(* CODESYS project AstroBROT.library
   Title: AstroBROT
   Version: 0.3.0
   Placeholder: AstroBROT
   Company: BROT

Project tree, tasks and I/O mapping:
  libraries: Tc2_Math, * (Beckhoff Automation GmbH); Tc2_Standard, * (Beckhoff Automation GmbH); Tc2_System, * (Beckhoff Automation GmbH); Tc2_Utilities, * (Beckhoff Automation GmbH); Tc3_Module, * (Beckhoff Automation GmbH)
  DUTs/
    data type E_TestState
  GVLs/
  POUs/
    FUNCTION_BLOCKS/
      function block FB_ALTAZ2HADEC [ST]
      function block FB_CO_ABERRATION [ST]
      function block FB_CO_NUTATE [ST]
      function block FB_CO_REFRACT [ST]
      function block FB_EQ2HOR [ST]
      function block FB_HADEC2ALTAZ [ST]
      function block FB_HOR2EQ [ST]
      function block FB_NUTATE [ST]
      function block FB_PRECESS [ST]
      function block FB_SUNPOS [ST]
    FUNCTIONS/
      function ATAN2 [ST]
      function CO_REFRACT_FORWARD [ST]
      function CT2LST [ST]
      function DateTime2JD [ST]
      function JD2LST [ST]
      function POLY [ST]
      function TEN [ST]
    program MAIN [ST]
  VISUs/
*)

// DUTs/E_TestState
{attribute 'qualified_only'}
{attribute 'strict'}
TYPE E_TestState :
(
	IDLE,
	EQ2HOR,
	HOR2EQ,
	EQ2EQ,
	JD2LST,
	ERROR
);
END_TYPE

// POUs/FUNCTION_BLOCKS/FB_ALTAZ2HADEC
FUNCTION_BLOCK FB_ALTAZ2HADEC
VAR_INPUT
	alt			: LREAL;	// the local apparent altitude, in DEGREES
	az			: LREAL;	// the local apparent azimuth, in DEGREES
	lat			: LREAL;	// the local geodetic latitude, in DEGREES
END_VAR
VAR_OUTPUT
	ha			: LREAL;	// the local apparent hour angle, in DEGREES
	dec			: LREAL;	// the local apparent declination, in DEGREES
END_VAR
VAR
	alt_r		: LREAL;
	az_r		: LREAL;
	lat_r		: LREAL;
	sindec		: LREAL;
END_VAR
VAR CONSTANT
	d2r			: LREAL := PI/180.0;
	r2d			: LREAL := 180.0/PI;
	//h2r:	LREAL := PI/12.0;
	//h2d:	LREAL := 15.0;
END_VAR

(*https://github.com/wlandsman/IDLAstro/blob/master/pro/

  NAME:
    ALTAZ2HADEC
 PURPOSE:
    Convert Horizon (Alt-Az) coordinates to Hour Angle and Declination.
 EXPLANATION::
    Can deal with the NCP singularity.    Intended mainly to be used by
    program hor2eq.pro
 CALLING SEQUENCE:
   ALTAZ2HADEC, alt, az, lat, ha, dec

 INPUTS
   alt - the local apparent altitude, in DEGREES, scalar or vector
   az  - the local apparent azimuth, in DEGREES, scalar or vector,
         measured EAST of NORTH!!!  If you have measured azimuth west-of-south
        (like the book MEEUS does), convert it to east of north via:
                       az = (az + 180) mod 360

   lat -  the local geodetic latitude, in DEGREES, scalar or vector.

 OUTPUTS
   ha  -  the local apparent hour angle, in DEGREES.  The hour angle is the 
          time that right ascension of 0 hours crosses the local meridian.  
          It is unambiguously defined.
   dec -  the local apparent declination, in DEGREES.

 EXAMPLE:
     Arcturus is observed at an apparent altitude of 59d,05m,10s and an 
     azimuth (measured east of north) of 133d,18m,29s while at the 
     latitude of +43.07833 degrees.
     What are the local hour angle and declination of this object?

     IDL> altaz2hadec, ten(59,05,10), ten(133,18,29), 43.07833, ha, dec
     ===> Hour angle ha = 336.683 degrees
          Declination, dec = 19.1824 degrees

       The widely available XEPHEM code gets:
                 Hour Angle = 336.683
                 Declination = 19.1824

 REVISION HISTORY:
    Written  Chris O'Dell Univ. of Wisconsin-Madison May 2002*)

alt_r  := alt*d2r;
az_r := az*d2r;
lat_r := lat*d2r;

//******************************************************************************
// find local HOUR ANGLE (in degrees, from 0. to 360.)
ha := atan2( (-SIN(az_r)*COS(alt_r)), (-COS(az_r)*SIN(lat_r)*COS(alt_r)+SIN(alt_r)*COS(lat_r)));
ha := ha / d2r;
IF ha < 0.0 THEN 
	ha := ha + 360.0;
END_IF
 ha := MODABS(ha, 360.0);

// Find declination (positive if north of Celestial Equator, negative if south)
sindec := SIN(lat_r)*SIN(alt_r) + COS(lat_r)*COS(alt_r)*COS(az_r);
// convert dec to degrees
dec := ASIN(sindec)/d2r;

END_FUNCTION_BLOCK

// POUs/FUNCTIONS/TEN
FUNCTION TEN : LREAL
VAR_INPUT
	dd, mm, ss	: LREAL;
END_VAR
VAR
END_VAR

TEN := dd + (mm/60.0) + (ss/3600.0);

END_FUNCTION

// POUs/FUNCTIONS/ATAN2
FUNCTION ATAN2 : LREAL
VAR_INPUT
	y		: LREAL;
	x		: LREAL;
END_VAR
VAR
END_VAR

(* source: https://de.wikipedia.org/wiki/Arctan2 *)
ATAN2 := 0.0;

IF x > 0 THEN
	ATAN2 := ATAN(y/x);
ELSIF x < 0 AND y > 0 THEN
	ATAN2 := ATAN(y/x) + PI;
ELSIF x < 0 AND y = 0 THEN
	ATAN2 := PI;
ELSIF x < 0 AND y < 0 THEN
	ATAN2 := ATAN(y/x) - PI;
ELSIF x = 0 AND y > 0 THEN
	ATAN2 := PI/2.0;
ELSIF x = 0 AND y < 0 THEN
	ATAN2 := -PI/2.0;
END_IF

END_FUNCTION

// POUs/FUNCTION_BLOCKS/FB_CO_ABERRATION
FUNCTION_BLOCK FB_CO_ABERRATION
VAR_INPUT
	jd			: LREAL;		// Julian Date
	ra			: LREAL;		// RA in degrees
	dec			: LREAL; 		// Dec in degrees
	eps 		: LREAL := 0.0;
END_VAR
VAR_OUTPUT
	d_ra		: LREAL;
	d_dec		: LREAL;
END_VAR
VAR
	sunpos		: FB_SUNPOS;
	nutate		: FB_NUTATE;
	sunra		: LREAL;
	sundec		: LREAL;
	sunlon		: LREAL;
	d_psi		: LREAL;
	d_epsilon	: LREAL; 
	eps0		: LREAL;
	t, e, peri, cd, sd, ce, te, cp, sp, cs, ss, ca, sa, term1, term2, term3, term4: LREAL;
END_VAR
VAR CONSTANT
	d2r 		: LREAL := PI/180.0;
	k			: LREAL := 20.49552; 	//constant of aberration, in arcseconds
	
END_VAR

(* https://github.com/wlandsman/IDLAstro/blob/master/pro/co_aberration.pro
;+
;  NAME:
;     CO_ABERRATION
; PURPOSE:
;     Calculate changes to Ra and Dec due to the effect of annual aberration 
; EXPLANATION:
;      as described in Meeus, Chap 23.
; CALLING SEQUENCE:
;      co_aberration, jd, ra, dec, d_ra, d_dec, [EPS = ]
; INPUTS
;       jd      : Julian Date [scalar or vector]
;       ra, dec : ra  and dec's in degrees
;
; OUTPUTS
;       d_ra, d_dec: the corrections to ra and dec due to aberration in 
;                    degrees.  (These values can be added to the true RA 
;                    and dec to get the apparent position).   Note that d_ra
;                     is *not* multiplied by cos(dec), so that 
;                     apparent_ra = ra + d_ra. 
; OPTIONAL INPUT KEYWORD:
;       eps : set this to the true obliquity of the ecliptic (in radians), or
;         it will be set for you if you don't know it (in that case, set it to
;                 an empty variable).
; NOTES:
;  These formula are from Meeus, Chapters 23.  Accuracy is much better than 1 
;   arcsecond.
;
;   The maximum deviation due to annual aberration is 20.49" and occurs when the
;   Earth velocity is perpendicular to the direction of the star.
;
; REVISION HISTORY:
;   Written, June 2002,      Chris O'Dell, U. of Wisconsin
;   Fix error with vector input   W. Landsman   June 2009
;   June 2009 update fixed case where JD was scalar but RA,Dec were vectors, but 
;     broke the case when both JD and RA,Dec were vectors Aug 2012 W. Landsman
;   Further fix when JD is 1 element vector  W. Landsman
;
;	UPDATE: HAS BEEN REWORKED FOR THE COORD STRUCTURE -> OUTPUT IS IN DEGREES
*)

T := (jd -2451545.0)/36525.0; // julian centuries from J2000 of jd.

IF eps = 0.0 THEN
	// must calculate obliquity of ecliptic
	nutate(jd := jd, nut_long => d_psi, nut_obliq => d_epsilon); //d_psi and d_epsilon in degrees
	eps0 := ten(23,26,21.448)*3600.0 - 46.8150*T - 0.00059*EXPT(T, 2) +  0.001813*EXPT(T, 3);
	// TRUE obliquity OF the ecliptic in radians
	eps := (eps0 + d_epsilon)/3600.0*d2r; 	
END_IF

sunpos(jd := jd, ra => sunra, dec => sundec, longmed => sunlon);

// Earth's orbital eccentricity
e := 0.016708634 - 0.000042037*T - 0.0000001267*EXPT(T, 2);
// longitude of perihelion, in degrees 
peri := 102.93735 + 1.71946*T + 0.00046*EXPT(T, 2);

//Useful Trig Functions
cd := COS(dec*d2r);		sd := SIN(dec*d2r);
ce := COS(eps); 		te := TAN(eps);
cp := COS(peri*d2r);	sp := SIN(peri*d2r);
cs := COS(sunlon*d2r);	ss := SIN(sunlon*d2r);
ca := COS(ra*d2r);		sa := SIN(ra*d2r);

term1 := (ca*cs*ce + sa*ss)/cd;
term2 := (ca*cp*ce + sa*sp)/cd;
term3 := (cs*ce*(te*cd - sa*sd) + ca*sd*ss);
term4 := (cp*ce*(te*cd - sa*sd) + ca*sd*sp);

d_ra := (-k * term1 + e*k * term2)/3600;
d_dec := (-k * term3 + e*k * term4)/3600;

END_FUNCTION_BLOCK

// POUs/FUNCTION_BLOCKS/FB_SUNPOS
FUNCTION_BLOCK FB_SUNPOS
VAR_INPUT
	jd				: LREAL;		// Julian Date
END_VAR
VAR_OUTPUT
	ra				: LREAL;		// right ascension
	dec				: LREAL;		// declination of the sun 
	longmed			: LREAL;		// longitude
	oblt			: LREAL;		// True Obliquity
END_VAR
VAR
	t				: LREAL;		//  Julian centuries FROM 1900.0
	l				: LREAL;		//  sun's mean longitude
	me				: LREAL;		// Earth's mean anomaly
	ellcor			: LREAL;		// ellipticity of the orbit
	mv				: LREAL;		// mean anomaly of Venus
	vencorr			: LREAL;		
	mm				: LREAL;		
	marscorr		: LREAL;		
	mj				: LREAL;		
	jupcorr			: LREAL;		
	d				: LREAL;		
	longterm		: LREAL;		
	mooncorr		: LREAL;		
	omega			: LREAL;
END_VAR
VAR CONSTANT
	d2r				: LREAL := PI/180.0; // Pi/180
END_VAR

(* https://github.com/wlandsman/IDLAstro/blob/master/pro/
NOTES:
;       Patrick Wallace (Rutherford Appleton Laboratory, UK) has tested the
;       accuracy of a C adaptation of the sunpos.pro code and found the 
;       following results.   From 1900-2100 SUNPOS  gave 7.3 arcsec maximum 
;       error, 2.6 arcsec RMS.  Over the shorter interval 1950-2050 the figures
;       were 6.4 arcsec max, 2.2 arcsec RMS.  
;
;       The returned ra and Dec are in the given date's equinox.
;
;       Procedure was extensively revised in May 1996, and the new calling
;       sequence is incompatible with the old one.source: https://idlastro.gsfc.nasa.gov/ftp/pro/astro/sunpos.pro *)

//  form TIME in Julian centuries FROM 1900.0
t := (jd - 2415020.0) / 36525.0;

//  form sun's mean longitude
l := (279.696678 + LMOD(36000.768925 * t, 360.0)) * 3600.0;

//  allow for ellipticity of the orbit (equation of centre) using the Earth's mean anomaly ME
me := 358.475844 + LMOD(35999.049750 * t, 360.0);
ellcor  := (6910.1 - 17.2 * t) * SIN(me * d2r) + 72.3 * SIN(2.0 * me*d2r);
l := l + ellcor;
 
// allow FOR the Venus perturbations using the mean anomaly OF Venus MV
mv := 212.603219 + LMOD(58517.803875 * t, 360.0);
vencorr := 4.8 * COS((299.1017 + mv - me)*d2r) + 
           5.5 * COS((148.3133 +  2.0 * mv  -  2.0 * me )*d2r) + 
           2.5 * COS((315.9433 +  2.0 * mv  -  3.0 * me )*d2r) + 
           1.6 * COS((345.2533 +  3.0 * mv  -  4.0 * me )*d2r) + 
           1.0 * COS((318.15   +  3.0 * mv  -  5.0 * me )*d2r);
l := l + vencorr;

//  Allow FOR the Mars perturbations using the mean anomaly OF Mars MM
mm := 319.529425  +  LMOD( 19139.858500 * t,  360.0 );
marscorr := 2.0 * COS((343.8883 -  2.0 * mm  +  2.0 * me)*d2r ) + 
            1.8 * COS((200.4017 -  2.0 * mm  + me) * d2r);
l := l + marscorr;

// Allow FOR the Jupiter perturbations using the mean anomaly OF Jupiter MJ
mj := 225.328328  +  LMOD( 3034.6920239 * t,  360.0 );
jupcorr := 7.2 * COS(( 179.5317 - mj + me )*d2r) + 
           2.6 * COS((263.2167  -  MJ ) *d2r) + 
           2.7 * COS(( 87.1450  -  2.0 * mj  +  2.0 * me ) *d2r) + 
           1.6 * COS((109.4933  -  2.0 * mj  +  me ) *d2r);
l := l + jupcorr;

// Allow FOR the Moons perturbations using the mean elongation OF the Moon from the Sun D
d := 350.7376814  + LMOD(445267.11422 * t,  360.0);
mooncorr  := 6.5 * SIN(d * d2r);
l := l + mooncorr;

// Allow for long period terms
longterm := 6.4 * SIN((231.19  +  20.20 * t) * d2r);
l :=  l + longterm;
l :=  LMOD(l + 2592000.0,  1296000.0); 
longmed := l / 3600.0;

// Allow for Aberration
l :=  l - 20.5;

// Allow for Nutation using the longitude of the Moons mean node OMEGA
omega := 259.183275 - LMOD(1934.142008 * t, 360.0);
l :=  l - 17.2 * SIN(omega * d2r);

// Form the True Obliquity
oblt := 23.452294 - 0.0130125 * t + (9.2 * COS(omega * d2r)) / 3600.0;

// Form Right Ascension AND Declination
l := l / 3600.0;
ra := ATAN2(SIN(l * d2r) * COS(oblt * d2r), COS(l * d2r));
dec := ASIN(SIN(l * d2r) * SIN(oblt * d2r));
 
ra := ra/d2r;
ra := MODABS(ra, 360.0);
dec := dec/d2r;

END_FUNCTION_BLOCK

// POUs/FUNCTION_BLOCKS/FB_NUTATE
FUNCTION_BLOCK FB_NUTATE
VAR_INPUT
	jd				: LREAL;			// Julian date
END_VAR
VAR_OUTPUT
	nut_long		: LREAL := 0.0;
	nut_obliq		: LREAL := 0.0;
END_VAR
VAR
	t				: LREAL;
	d, M, Mprime, F, omega: LREAL;
	arg, sarg, carg	: ARRAY[0..62] OF LREAL;
	I				: INT;
END_VAR
VAR CONSTANT
	d2r				: LREAL := PI/180.0;
	coeff1			: ARRAY[0..3] OF LREAL := [297.85036, 445267.111480, -0.0019142,  1.0/189474];
	coeff2			: ARRAY[0..3] OF LREAL := [357.52772,  35999.050340, -0.0001603, -1.0/3E5]; 
	coeff3			: ARRAY[0..3] OF LREAL := [134.96298, 477198.867398,  0.0086972,  1.0/5.625E4]; 
	coeff4			: ARRAY[0..3] OF LREAL :=  [93.27191, 483202.017538, -0.0036825, -1.0/3.27270E5]; 
  	coeff5			: ARRAY[0..3] OF LREAL := [125.04452,  -1934.136261,  0.0020708,  1.0/4.5E5];
	d_lng			: ARRAY[0..62] OF LREAL := [0,-2,0,0,0,0,-2,0,0,-2,-2,-2,0,2,0,2,0,0,-2,0,2,0,0,-2,0,-2,0,0,2,-2,0,-2,0,0,2,2,0,-2,0,2,2,-2,-2,2,2,0,-2,-2,0,-2,-2,0,-1,-2,1,0,0,-1,0,0,2,0,2]; 
	m_lng			: ARRAY[0..62] OF LREAL := [0,0,0,0,1,0,1,0,0,-1,17(0),2,0,2,1,0,-1,0,0,0,1,1,-1,0,0,0,0,0,0,-1,-1,0,0,0,1,0,0,1,0,0,0,-1,1,-1,-1,0,-1];
	mp_lng			: ARRAY[0..62] OF LREAL := [0,0,0,0,0,1,0,0,1,0,1,0,-1,0,1,-1,-1,1,2,-2,0,2,2,1,0,0,-1,0,-1,0,0,1,0,2,-1,1,0,1,0,0,1,2,1,-2,0,1,0,0,2,2,0,1,1,0,0,1,-2,1,1,1,-1,3,0];
	f_lng			: ARRAY[0..62] OF LREAL := [0,2,2,0,0,0,2,2,2,2,0,2,2,0,0,2,0,2,0,2,2,2,0,2,2,2,2,0,0,2,0,0,0,-2,2,2,2,0,2,2,0,2,2,0,0,0,2,0,2,0,2,-2,0,0,0,2,2,0,0,2,2,2,2];
	om_lng			: ARRAY[0..62] OF LREAL := [1,2,2,2,0,0,2,1,2,2,0,1,2,0,1,2,1,1,0,1,2,2,0,2,0,0,1,0,1,2,1,1,1,0,1,2,2,0,2,1,0,2,1,1,1,0,1,1,1,1,1,0,0,0,0,0,2,0,0,2,2,2,2];
	sin_lng			: ARRAY[0..62] OF LREAL := [-171996, -13187, -2274, 2062, 1426, 712, -517, -386, -301, 217, -158, 129, 123, 63, 63, -59, -58, -51, 48, 46, -38, -31, 29, 29, 26, -22, 21, 17, 16, -16, -15, -13, -12, 11, -10, -8, 7, -7, -7, -7, 6,6,6,-6,-6,5,-5,-5,-5,4,4,4,-4,-4,-4,3,-3,-3,-3,-3,-3,-3,-3 ];
	sdelt			: ARRAY[0..62] OF LREAL := [-174.2, -1.6, -0.2, 0.2, -3.4, 0.1, 1.2, -0.4, 0, -0.5, 0, 0.1, 0,0,0.1, 0,-0.1,10(0), -0.1, 0, 0.1, 33(0)];
	cos_lng			: ARRAY[0..62] OF LREAL := [ 92025, 5736, 977, -895, 54, -7, 224, 200, 129, -95,0,-70,-53,0, -33, 26, 32, 27, 0, -24, 16,13,0,-12,0,0,-10,0,-8,7,9,7,6,0,5,3,-3,0,3,3, 0,-3,-3,3,3,0,3,3,3, 14(0)] ;
	cdelt			: ARRAY[0..62] OF LREAL := [8.9, -3.1, -0.5, 0.5, -0.1, 0.0, -0.6, 0.0, -0.1, 0.3, 53(0)];
END_VAR

//https://github.com/wlandsman/IDLAstro/blob/master/pro/nutate.pro
(*METHOD:
;       Uses the formula in Chapter 22 of ``Astronomical Algorithms'' by Jean 
;       Meeus (1998, 2nd ed.) which is based on the 1980 IAU Theory of Nutation
;       and includes all terms larger than 0.0003".*)

//  form time in Julian centuries from 1900.0

t := (jd - 2451545.0)/36525.0;

// Mean elongation of the Moon

d := poly(T, coeff1)*d2r;
d := MODABS(d, 2.0*PI);

// Sun's mean anomaly

M := poly(T,coeff2)*d2r;
M := MODABS(M, 2.0*PI);

// Moon's mean anomaly

Mprime := poly(T,coeff3)*d2r;
Mprime := MODABS(Mprime, 2.0*PI);

// Moon's argument of latitude

F := poly(T, coeff4 )*d2r;
F := MODABS(F, 2.0*PI);

// Longitude OF the ascending node OF the Moon's mean orbit on the ecliptic,
//  measured from the mean equinox of the date

omega := poly(T, coeff5)*d2r;
omega := MODABS(omega, 2.0*PI);


// Sum the periodic terms 
FOR i:=0 TO 62 DO
	arg[i] := d_lng[i]*d + m_lng[i]*m +mp_lng[i]*mprime + f_lng[i]*f +om_lng[i]*omega;
	sarg[i] := SIN(arg[i]);
	carg[i] := COS(arg[i]);
END_FOR

nut_long  := 0.0;
nut_obliq := 0.0;

FOR i:=0 TO 62 DO
	nut_long  := nut_long  + 0.0001*( (sdelt[i]*t + sin_lng[i])*sarg[i]);
	nut_obliq := nut_obliq + 0.0001*( (cdelt[i]*t + cos_lng[i])*carg[i]);
END_FOR

END_FUNCTION_BLOCK

// POUs/FUNCTIONS/POLY
FUNCTION POLY : LREAL
VAR_INPUT
	X			: LREAL;
	COEFFS		: ARRAY [0..3] OF LREAL;
END_VAR
VAR
END_VAR

POLY := COEFFS[0]*EXPT(X, 0) + COEFFS[1]*EXPT(X, 1) + COEFFS[2]*EXPT(X, 2) + COEFFS[3]*EXPT(X, 3);

END_FUNCTION

// POUs/FUNCTION_BLOCKS/FB_CO_NUTATE
FUNCTION_BLOCK FB_CO_NUTATE
VAR_INPUT
	jd			: LREAL;		// Julian date
	ra			: LREAL;		// RA in degrees
	dec			: LREAL;		// Dec in degrees
END_VAR
VAR_OUTPUT
	d_ra		: LREAL;		// RA diff in degrees
	d_dec		: LREAL;		// Dec diff in degrees
	eps			: LREAL;		// TRUE obliquity OF the ecliptic in radians
	d_psi		: LREAL;		// in arcsec
	d_eps		: LREAL;
END_VAR
VAR
	T, eps0, ce, se,x,y,z,x2,y2,z2,rad,xyproj,ra2,dec2: LREAL;
	nutate		: FB_NUTATE;
END_VAR
VAR CONSTANT
	d2r			: LREAL := PI/180.0;
	d2as		: LREAL := PI/(180.0*3600.0);
END_VAR

// https://github.com/wlandsman/IDLAstro/blob/master/pro/co_nutate.pro
(*EXPLANATION:
;     Calculates necessary changes to ra and dec due to
;     the nutation of the Earth's rotation axis, as described in Meeus, Chap 23.
;     Uses formulae from Astronomical Almanac, 1984, and does the calculations
;     in equatorial rectangular coordinates to avoid singularities at the
;     celestial poles.*)
// Julian centuries FROM J2000 OF jd.
T := (jd -2451545.0)/36525.0; 

// must calculate obliquity OF ecliptic
nutate(jd := jd,
		nut_long => d_psi, 
		nut_obliq => d_eps); 

eps0 := 23.4392911*3600.0 - 46.8150*T - 0.00059*EXPT(T, 2) + 0.001813*EXPT(T, 3);
eps := (eps0 + d_eps)/3600.0*d2r; // TRUE obliquity OF the ecliptic in radians
 
//useful numbers
ce := COS(eps);
se := SIN(eps);

// convert ra-dec to equatorial rectangular coordinates
x := COS(ra*d2r) * COS(dec*d2r);
y := SIN(ra*d2r) * COS(dec*d2r);
z := SIN(dec*d2r);

// apply corrections to each rectangular coordinate
x2 := x - (y*ce + z*se)*d_psi * d2as;
y2 := y + (x*ce*d_psi - z*d_eps) * d2as;
z2 := z + (x*se*d_psi + y*d_eps) * d2as;

// convert back to equatorial spherical coordinates
rad := SQRT(x2*x2 + y2*y2 + z2*z2);
xyproj := SQRT(x2*x2 + y2*y2);

ra2  := x2 * 0.0;
dec2 := x2 * 0.0;

// Calculate Ra and Dec in RADIANS (later convert to DEGREES)
IF (xyproj = 0) AND (z <> 0) THEN
	// places where xyproj=0 (point at NCP or SCP)
	dec2 := ASIN(z2/rad);
	ra2 := 0.0;
END_IF
 
IF (xyproj <> 0) THEN
	// places other than NCP or SCP
	ra2 := ATAN2(y2, x2);
	dec2 := ASIN(z2/rad);
END_IF

// convert to DEGREES

ra2 := ra2 /d2r;
dec2 := dec2 /d2r;

ra2 := MODABS(ra2, 360.0);


// Return changes in ra and dec
d_ra := (ra2 - ra);
d_dec := (dec2 - dec);

END_FUNCTION_BLOCK

// POUs/FUNCTION_BLOCKS/FB_CO_REFRACT
FUNCTION_BLOCK FB_CO_REFRACT
VAR_INPUT
	old_alt			: LREAL;			// old alt in degrees
	altitude		: LREAL := 0.0;		// altitude of observatory
	pressure		: LREAL := 0.0;		// pressure
	temperature		: LREAL := 0.0;		// temperature
	epsilon			: LREAL := 0.25; 	//accuracy of iteration for observed=TRUE case, in arcseconds
	TO_OBSERVED		: BOOL;
END_VAR
VAR_OUTPUT
	new_alt			: LREAL;
END_VAR
VAR
	aout, P, T, dr, cur, last : LREAL;
END_VAR
VAR CONSTANT
	alpha 			: LREAL := 0.0065; 	//temp lapse rate [deg C per meter]
END_VAR

// https://github.com/wlandsman/IDLAstro/blob/master/pro/co_refract.pro
IF temperature = 0.0 THEN
	IF altitude > 11000.0 THEN 
		temperature := 211.5; 
	ELSE 
		temperature := 283.0 - alpha*altitude;
	END_IF
END_IF

// estimate Pressure based on altitude, using U.S. Standard Atmosphere formula.
IF pressure = 0 THEN 
	pressure := 1010.0*EXPT(1-6.5/288000*altitude, 5.255);
END_IF

IF NOT TO_OBSERVED THEN 
	aout := old_alt - co_refract_forward(old_alt, P:=pressure,T:=temperature);
ELSE
	aout := 0.0;
	P := pressure; T := temperature;
	//calculate initial refraction guess
	dr := co_refract_forward(old_alt, P:=P, T:=T);
	cur := old_alt + dr; // guess of observed location

	REPEAT 
	 	last := cur;
		dr := co_refract_forward(cur, P:= P, T:=T);
	  	cur := old_alt + dr;
	UNTIL ABS(last-cur)*3600.0 < epsilon
	END_REPEAT
	aout := cur;
END_IF

new_alt := aout;

END_FUNCTION_BLOCK

// POUs/FUNCTIONS/CO_REFRACT_FORWARD
FUNCTION CO_REFRACT_FORWARD : LREAL
VAR_INPUT
	a			: LREAL; 			// The observed (apparent) altitude, in DEGREES.
	P			: LREAL := 1010.0;	// Pressure [in millibars]. Default is 1010 millibars.
	T			: LREAL := 0.0;		// Ground Temp [in Celsius].  Default is 0 Celsius.
END_VAR
VAR
	ref			: LREAL;
	tpcor		: LREAL;
END_VAR
VAR CONSTANT
	d2r 		: LREAL := PI/180.0;
END_VAR

a := LIMIT(0.0, a, 90.0);
P := LIMIT(600.0, P, 1200.0);
T := LIMIT(-40.0, T, 40.0);

IF a >= 15.0 THEN
	ref := 1.0 / TAN((a + 7.31 / (a + 4.4)) * d2r);
ELSE
	ref := 3.569 * (0.1594 + 0.0196 * a + 0.00002 * EXPT(a, 2)) / (1.0 + 0.505 * a + 0.0845 * EXPT(a, 2));
END_IF
tpcor := P * 283.15 / (1010.0 * (273.15 + T));
CO_REFRACT_FORWARD := tpcor * ref;

END_FUNCTION

// POUs/FUNCTION_BLOCKS/FB_EQ2HOR
FUNCTION_BLOCK FB_EQ2HOR
VAR_INPUT
	ra				: LREAL;	// right ascension in degrees
	dec				: LREAL;	// declination in degrees
	jd				: LREAL;	// Julian Date
	lon				: LREAL;	// longitude in degrees
	lat				: LREAL;	// latitude in degrees
	ws				: BOOL := FALSE; 	// Set this to TRUE get the azimuth measured westward FROM south (NOT East of North).
	precess			: BOOL := TRUE; 	// Set this to 1 to force precession [default], 0 for no precession correction
	nutate			: BOOL := TRUE; 	// Set this to 1 to force nutation [default], 0 for no nutation correction.
	aberration		: BOOL := TRUE; 	// Set this to 1 to force aberration correction [default], 0 for no correction.
	refract 		: BOOL := TRUE; 	// Set to 1 to force refraction correction[default] (for actual sky coord), 0 for no correction (for theoretical coord).
	refract_to_observed : BOOL := TRUE;
	altitude		: LREAL := 0.0;
END_VAR
VAR_OUTPUT
	alt				: LREAL;		// altitude in degrees
	az				: LREAL;		// azimuth in degrees
	ha				: LREAL;		// hour angle in degreesss
END_VAR
VAR
	tstart, J_now	: LREAL;
	lmst			: LREAL;
	last			: LREAL;
	d_psi			: LREAL;
	eps				: LREAL;
	fbprecess		: FB_PRECESS;
	hadec2altaz		: FB_HADEC2ALTAZ;
	co_nutate		: FB_CO_NUTATE;
	co_aberration	: FB_CO_ABERRATION;
	co_refract		: FB_CO_REFRACT;
	ra_pre			: LREAL;		// Precessed RA in degrees
	dec_pre			: LREAL;		// Precessed Dec in degrees
	d_ra_abr		: LREAL;		// Difference in RA due to aberration
	d_dec_abr		: LREAL;		// Difference in Dec due to aberration
	d_ra_nut		: LREAL;		// Difference in RA due to nutation
	d_dec_nut		: LREAL;		// Difference in Dec due to nutation
END_VAR
VAR CONSTANT
	// easier then functions
	d2r				: LREAL := PI/180.0;
	h2r				: LREAL := PI/12.0;
	jd2000			: LREAL := 2451545.0;
END_VAR

(* source https://github.com/wlandsman/IDLAstro/blob/master/pro/eq2hor.pro 

PURPOSE:
	Convert celestial  (ra-dec) coords to local horizon coords (alt-az).

DESCRIPTION:
This  code calculates horizon (alt,az) coordinates from equatorial
(ra,dec) coords. It is typically accurate to about 1 arcsecond or better (I
have checked the output against the publicly available XEPHEM software). It
performs precession, nutation, aberration, and refraction corrections. [...]
*)


tstart := 2000.0;

(* ******************************************************************************
 PRECESS coordinates to current date
 (uses astro lib procedure PRECESS.pro)
*)
J_now := (JD - jd2000)/365.25 + 2000.0; // compute current equinox
IF precess THEN
	fbprecess( 
		ra := ra, 
		dec := dec, 
		equinox1 := tstart, 
		equinox2 := J_now, 
		ra_precessed => ra_pre, 
		dec_precessed => dec_pre);
ELSE
	ra_pre := ra;
	dec_pre := dec;
END_IF

(******************************************************************************
 calculate NUTATION and ABERRATION Corrections to Ra-Dec 
*)

IF nutate THEN
	co_nutate(	
		jd := jd, 
		ra := ra_pre, 
		dec := dec_pre, 
		d_ra => d_ra_nut, 
		d_dec => d_dec_nut,
		eps=>eps, 
		d_psi=>d_psi);
END_IF

IF ABERRATION THEN	
	co_aberration(	
		jd := jd, 
		ra := ra_pre, 
		dec := dec_pre, 
		d_ra => d_ra_abr, 
		d_dec => d_dec_abr,
		eps := eps);	
END_IF
ra := ra_pre + d_ra_abr + d_ra_nut;
dec := dec_pre + d_dec_abr + d_dec_nut;

(***************************************************************************************
Calculate LOCAL MEAN SIDEREAL TIME *)
lmst := jd2lst(JD:=jd, lon:=lon);
// calculate local APPARENT sidereal time
last := lmst + d_psi *COS(eps)/3600.0 ; //add correction in degrees

(******************************************************************************
 Find hour angle (in DEGREES) *)
ha := last - ra;
ha := MODABS(ha, 360.0);

(*******************************************************************************
 Now do the spherical trig to get APPARENT alt,az. *)
hadec2altaz(	
	ha := ha, 
	dec := dec, 
	lat := lat, 
	alt => alt, 
	az => az, 
	WS := WS);

(********************************************************************************************
 Make Correction for ATMOSPHERIC REFRACTION
 (use this for visible and radio wavelengths; author is unsure about other wavelengths.
  See the comments in CO_REFRACT for more details.) *)
IF refract THEN 
	co_refract(	
		old_alt := alt, 
		altitude := altitude, 
		to_observed := refract_to_observed, 
		new_alt => alt);
END_IF

END_FUNCTION_BLOCK

// POUs/FUNCTIONS/JD2LST
FUNCTION JD2LST : LREAL
VAR_INPUT
	jd			: LREAL;	// Julian date
	lon			: LREAL;	// longitude in degrees
END_VAR
VAR
	T			: LREAL;
	theta0		: LREAL;
END_VAR
VAR CONSTANT
	jd2000		: LREAL := 2451545.0;
END_VAR

// following https://squarewidget.com/astronomical-calculations-sidereal-time/
T := ((jd - jd2000) / 36525.0);
theta0 := 280.46061837 + 360.98564736629 * (JD - jd2000) + (0.000387933 * T * T) - (T * T * T / 38710000.0); // (12.4)

// LST is only defined from 0 to 360
JD2LST := MODABS(theta0 + lon, 360.0); // LST in degrees

END_FUNCTION

// POUs/FUNCTION_BLOCKS/FB_PRECESS
FUNCTION_BLOCK FB_PRECESS
VAR_INPUT
	ra				: LREAL;		// RA in degrees
	dec				: LREAL;		// Dec in degrees
	equinox1		: LREAL;
	equinox2		: LREAL;
END_VAR
VAR_OUTPUT
	ra_precessed	: LREAL;
	dec_precessed	: LREAL;
END_VAR
VAR
	ra_rad			: LREAL;		// RA in rad
	dec_rad			: LREAL;		// Dec in rad
	a, b, c, t		: LREAL;
	x, x2			: ARRAY[0..2] OF LREAL;
	st1				: LREAL;
	rot				: ARRAY[0..2,0..2] OF LREAL;
	sina, sinb, sinc, cosa,cosb,cosc: LREAL;
END_VAR
VAR CONSTANT
	d2r 			: LREAL := PI/180.0;
	sec_to_rad 		: LREAL := d2r/3600.0;
END_VAR

//https://github.com/wlandsman/IDLAstro/blob/master/pro/precess.pro

(*
; RESTRICTIONS:
;       Accuracy of precession decreases for declination values near 90 
;       degrees.  PRECESS should not be used more than 2.5 centuries from
;       2000 on the FK5 system (1950.0 on the FK4 system).
; PROCEDURE:
;       Algorithm from Computational Spherical Astronomy by Taff (1983), 
;       p. 24. (FK4). FK5 constants from "Astronomical Almanac Explanatory
;       Supplement 1992, page 104 Table 3.211.1.
*)

// deg 2 radian
ra_rad := ra*d2r;
dec_rad := dec*d2r;


a := COS( dec_rad );
x[0] := a*COS(ra_rad); x[1] := a*SIN(ra_rad); x[2] := SIN(dec_rad);

//*** PREMAT code starts here
ST1 := 0.001*( equinox1 - 2000.0);
t := 0.001*( equinox2 - equinox1);
//  Compute 3 rotation angles
A := sec_to_rad * T * (23062.181 + ST1*(139.656 +0.0139*ST1) + T*(30.188 - 0.344*ST1+17.998*T));
B := sec_to_rad * T * T * (79.280 + 0.410*ST1 + 0.205*T) + A;
C := sec_to_rad * T * (20043.109 - ST1*(85.33 + 0.217*ST1) + T*(-42.665 - 0.217*ST1 -41.833*T));
  sina := SIN(a); sinb := SIN(b);  sinc := SIN(c);
  cosa := COS(a); cosb := COS(b);  cosc := COS(c);

rot[0,0] :=  cosa*cosb*cosc-sina*sinb; 	rot[0,1] := sina*cosb+cosa*sinb*cosc; 	rot[0,2] := cosa*sinc;
rot[1,0] := -cosa*sinb-sina*cosb*cosc; 	rot[1,1] := cosa*cosb-sina*sinb*cosc; 	rot[1,2] := -sina*sinc;
rot[2,0] := -cosb*sinc;					rot[2,1] := -sinb*sinc; 				rot[2,2] := cosc;

//*** PREMAT code ends here

//x2 := rot* x; //rotate to get output direction cosines
x2[0] := rot[0,0]*x[0] + rot[1,0]*x[1] + rot[2,0]*x[2];
x2[1] := rot[0,1]*x[0] + rot[1,1]*x[1] + rot[2,1]*x[2];
x2[2] := rot[0,2]*x[0] + rot[1,2]*x[1] + rot[2,2]*x[2];

ra_rad := atan2(x2[1],x2[0]);
dec_rad := ASIN(x2[2]);

ra_precessed := ra_rad/d2r;
ra_precessed := MODABS(ra_precessed, 360.0);            //RA between 0 AND 360 degrees
dec_precessed := dec_rad/d2r;

END_FUNCTION_BLOCK

// POUs/FUNCTION_BLOCKS/FB_HADEC2ALTAZ
FUNCTION_BLOCK FB_HADEC2ALTAZ
VAR_INPUT
	ha				: LREAL;		// Hour angle in degrees
	dec				: LREAL;		// Declination in degrees
	lat				: LREAL;		// Latitude in degrees
	WS				: BOOL := FALSE;
END_VAR
VAR_OUTPUT
	alt				: LREAL;		// altitude in degrees
	az				: LREAL;		// azimuth in degrees
END_VAR
VAR
	sh,sd,sl, ch,cd,cl,	x, y, z, radius: LREAL;
END_VAR
VAR CONSTANT
	d2r 			: LREAL := PI/180.0;
END_VAR

(* source https://github.com/wlandsman/IDLAstro/blob/master/pro/hadec2altaz.pro
;+
;  NAME:
;     HADEC2ALTAZ
;  PURPOSE:
;      Converts Hour Angle and Declination to Horizon (alt-az) coordinates.
;  EXPLANATION:
;      Can deal with NCP/SCP singularity.    Intended mainly to be used by
;      program EQ2HOR
;
; CALLING SEQUENCE:
;      HADEC2ALTAZ, ha, dec, lat ,alt ,az [ /WS ]
;
; INPUTS
;     ha -  the local apparent hour angle, in DEGREES, scalar or vector
;     dec -  the local apparent declination, in DEGREES, scalar or vector
;     lat -  the local latitude, in DEGREES, scalar or vector
;
; OUTPUTS
;     alt - the local apparent altitude, in DEGREES.
;     az  - the local apparent azimuth, in DEGREES, all results in double
;           precision
; OPTIONAL KEYWORD INPUT:
;      /WS - Set this keyword for the output azimuth to be measured West from 
;            South.    The default is to measure azimuth East from North.
;
; EXAMPLE:
;     What were the apparent altitude and azimuth of the sun when it transited 
;     the local meridian at Pine Bluff Observatory (Lat=+43.07833 degrees) on 
;     April 21, 2002?   An object transits the local meridian at 0 hour angle.
;     Assume this will happen at roughly 1 PM local time (18:00 UTC).
;
;     IDL> jdcnv, 2002, 4, 21, 18., jd  ; get rough Julian date to determine 
;                                       ;Sun ra, dec.
;     IDL> sunpos, jd, ra, dec
;     IDL> hadec2altaz, 0., dec, 43.078333, alt, az
;
;       ===> Altitude alt = 58.90
;            Azimuth  az = 180.0

; REVISION HISTORY:
;      Written  Chris O'Dell Univ. of Wisconsin-Madison May 2002
;-
*)
sh := SIN(ha*d2r);
ch := COS(ha*d2r);
sd := SIN(dec*d2r);
cd := COS(dec*d2r);
sl := SIN(lat*d2r);
cl := COS(lat*d2r);

x := -ch * cd * sl + sd * cl;
y := -sh * cd;
z := ch * cd * cl + sd * sl;
radius := SQRT(x*x + y*y);

// now get Alt, Az
az := ATAN2(y, x) /d2r;	// was ATAN(y, x)
alt := ATAN2(z, radius) / d2r;

// correct for negative AZ
az := MODABS(az, 360.0);

// convert AZ to West from South, if desired
IF WS THEN 
	az := MODABS(az + 180.0, 360);
END_IF

END_FUNCTION_BLOCK

// POUs/FUNCTION_BLOCKS/FB_HOR2EQ
FUNCTION_BLOCK FB_HOR2EQ
VAR_INPUT
	alt				: LREAL;			//altitude (in degrees)  
	az				: LREAL;			//azimuth angle (in degrees, measured EAST from NORTH, but see keyword WS below.) [scalar or vector]
	jd				: LREAL;			// Julian Date
	lat				: LREAL;			// observers latitude (degrees)
	lon				: LREAL;			// observers longitude (degrees)
	ws				: BOOL := FALSE; 	// Set this to TRUE get the azimuth measured westward FROM south (NOT East of North).
	precess			: BOOL := TRUE; 	// Set this to 1 to force precession [default], 0 for no precession correction
	nutate			: BOOL := TRUE; 	// Set this to 1 to force nutation [default], 0 for no nutation correction.
	aberration		: BOOL := TRUE; 	// Set this to 1 to force aberration correction [default], 0 for no correction.
	refract			: BOOL := TRUE; 	// Set to 1 to force refraction correction[default] (for actual sky coord), 0 for no correction (for theoretical coord).
	altitude		: LREAL := 0.0;
	refract_to_observed : BOOL := TRUE;
END_VAR
VAR_OUTPUT
	ra				: LREAL;			// Right Ascension of object  (J2000) in degrees (FK5)
	dec				: LREAL;			// Declination of object (J2000) in degrees (FK5)
	ha				: LREAL;			// hour angle (in degrees) (optional)
END_VAR
VAR
	lmst			: LREAL;
	J_now			: LREAL;
	co_nutate		: FB_CO_NUTATE;
	co_aberration	: FB_CO_ABERRATION;
	co_refract		: FB_CO_REFRACT;
	fbprecess		: FB_PRECESS;
	altaz2hadec		: FB_ALTAZ2HADEC;
	last			: LREAL;
	eps				: LREAL;
	d_psi			: LREAL;
	d_ra_abr		: LREAL;		// Difference in RA due to aberration
	d_dec_abr		: LREAL;		// Difference in Dec due to aberration
	d_ra_nut		: LREAL;		// Difference in RA due to nutation
	d_dec_nut		: LREAL;		// Difference in Dec due to nutation
	d_ra_ref		: LREAL;		// time reference
	d_dec_ref		: LREAL;		// time reference
END_VAR
VAR CONSTANT
	// easier then functions
	d2r				: LREAL := PI/180.0;
	h2d				: LREAL := 15.0;
	jd2000			: LREAL := 2451545.0;
END_VAR

(* https://github.com/wlandsman/IDLAstro/blob/master/pro/hor2eq.pro
; NAME:
;   HOR2EQ
;
; PURPOSE:
;    Converts local horizon coords (alt-az) of something to equatorial (ra-dec).
;
; EXPLANATION:
;     This is a nice code to calculate equatorial (ra,dec) coordinates from
;     horizon (alt,az) coords.    It is typically accurate to about 1 arcsecond
;     or better (I have checked the output against the publicly available XEPHEM
;     software). It performs precession, nutation, aberration, and refraction
;     corrections.  The perhaps best thing about it is that it can take arrays
;     as inputs, in all variables and keywords EXCEPT Lat, lon, and Altitude
;    (the code assumes these aren't changing), and uses vector arithmetic in
;     every calculation except when calculating the precession matrices.
;
; DEPENDENCIES:
;       NUTATE, PRECESS, SUNPOS,
;       CO_NUTATE, CO_ABERRATION, CO_REFRACT, HADEC2ALTAZ
;CORRECTIONS I DO NOT MAKE:
;   *  Deflection of Light by the sun due to GR. (typically milliarcseconds,
;        can be arcseconds within one degree of the sun)
;   *  The Effect of Annual Parallax (typically < 1 arcsecond)
;   *  and more (see below)
;
; TO DO
;    * Better Refraction Correction.  Need to put in wavelength dependence,
;       and integrate through the atmosphere.
;    * Topocentric Parallax Correction (will take into account elevation of
;          the observatory)
;    * Proper Motion (but this will require crazy lookup tables or something).
;    * Difference between UTC and UT1 in determining LAST -- is this important?
;    * Effect of Annual Parallax (is this the same as topocentric Parallax?)
;    * Polar Motion
;    * Better connection to Julian Date Calculator.
;
; AUTHOR:
;   Chris O'Dell
;   Assistant Professor of Atmospheric Science
;   Colorado State University
;   Email: odell@atmos.colostate.edu
; REVISION HISTORY:
;     Made all integers type LONG  W. Landsman   September 2007
;     Fixed for case of scalar Julian date but vector positions W L June 2009
;-*)

IF WS THEN 
	az := az - 180.0;
END_IF

(********************************************************************************************
 Make Correction for ATMOSPHERIC REFRACTION
 (use this for visible and radio wavelengths; author is unsure about other wavelengths.
  See the comments in CO_REFRACT for more details.) *)
IF refract THEN 
	co_refract(	
		old_alt := alt, 
		altitude := altitude, 
		to_observed := refract_to_observed, 
		new_alt => alt);
END_IF


//******************************************************************************
//Calculate LOCAL APPARENT SIDEREAL TIME
// Nutation for d_psi and eps
co_nutate(
	jd := jd, 
	ra := 45.0, 
	dec := 45.0, 
	d_ra => d_ra_nut, 
	d_dec => d_dec_nut,  
	eps=>eps, 
	d_psi=>d_psi);
// first get local mean sidereal time (lmst)
// get LST (in hours) - note:this is indep of tzone since giving jd
// Calculate LOCAL MEAN SIDEREAL TIME 
lmst := jd2lst(JD:=jd, lon:=lon);
// calculate local APPARENT sidereal time
last := lmst + d_psi *COS(eps)/3600.0 ; //add correction in degrees


//****************************************************************************
// Now do the spherical trig to get APPARENT Hour Angle [degrees], and
// declination [degrees].
altaz2hadec(alt := alt, az := az, lat := lat, ha => ha, dec => dec);

// Find Right Ascension (in degrees, from 0 to 360.)
ra := MODABS(last - ha + 360.0, 360.0);

//*****************************************************************************
// calculate NUTATION and ABERRATION Corrections to Ra-Dec
IF nutate THEN
	co_nutate(	
		jd := jd, 
		ra := ra, 
		dec := dec, 
		d_ra => d_ra_nut, 
		d_dec => d_dec_nut, 
		eps=>eps, 
		d_psi=>d_psi);
END_IF
IF ABERRATION THEN	
	co_aberration(	
		jd := jd, 
		ra := ra, 
		dec := dec,
		eps := eps,
		d_ra => d_ra_abr, 
		d_dec => d_dec_abr);
END_IF
ra := ra - (d_ra_abr + d_ra_nut);
dec := dec - (d_dec_abr + d_dec_nut);
 


(* ******************************************************************************
 PRECESS coordinates to current date
 (uses astro lib procedure PRECESS.pro)
*)
J_now := (jd - jd2000)/365.25 + 2000.0; // compute current equinox
IF precess THEN
	fbprecess( 
		ra := ra, 
		dec := dec, 
		equinox1 := J_now, 
		equinox2 := 2000.0, 
		ra_precessed => ra, 
		dec_precessed => dec);
END_IF

END_FUNCTION_BLOCK

// POUs/FUNCTIONS/CT2LST
FUNCTION CT2LST : LREAL
VAR_INPUT
	lng: LREAL; // The longitude in degrees (east of Greenwich) of the place for which the local sidereal time is desired, scalar.   The Greenwich mean sidereal time (GMST) can be found by setting Lng = 0.
	jd:	LREAL; // this is the Julian date of time in question
END_VAR
VAR
	t0,t,theta: LREAL;
END_VAR
VAR CONSTANT
	jd2000: LREAL := 2451545.0;
END_VAR

(* https://github.com/wlandsman/IDLAstro/blob/master/pro/ct2lst.pro 

;+
; NAME:
;     CT2LST
; PURPOSE:
;     To convert from Local Civil Time to Local Mean Sidereal Time.
;
; CALLING SEQUENCE:
;     CT2LST, Lst, Lng, Tz, Time, [Day, Mon, Year] 
;                       or
;     CT2LST, Lst, Lng, dummy, JD
;
; INPUTS:
;     Lng  - The longitude in degrees (east of Greenwich) of the place for 
;            which the local sidereal time is desired, scalar.   The Greenwich 
;            mean sidereal time (GMST) can be found by setting Lng = 0.
;     Tz  - The time zone of the site in hours, positive East  of the Greenwich
;           meridian (ahead of GMT).  Use this parameter to easily account 
;           for Daylight Savings time (e.g. -4=EDT, -5 = EST/CDT), scalar
;           This parameter is not needed (and ignored) if Julian date is 
;           supplied.    ***Note that the sign of TZ was changed in July 2008
;           to match the standard definition.*** 
;     Time or JD  - If more than four parameters are specified, then this is 
;               the time of day of the specified date in decimal hours.  If 
;               exactly four parameters are specified, then this is the 
;               Julian date of time in question, scalar or vector
;
; OPTIONAL INPUTS:
;      Day -  The day of the month (1-31),integer scalar or vector
;      Mon -  The month, in numerical format (1-12), integer scalar or vector
;      Year - The 4 digit year (e.g. 2008), integer scalar or vector
;
; OUTPUTS:
;       Lst   The Local Sidereal Time for the date/time specified in hours.
;
; RESTRICTIONS:
;       If specified, the date should be in numerical form.  The year should
;       appear as yyyy.
;
; PROCEDURE:
;       The Julian date of the day and time is question is used to determine
;       the number of days to have passed since 0 Jan 2000.  This is used
;       in conjunction with the GST of that date to extrapolate to the current
;       GST; this is then used to get the LST.    See Astronomical Algorithms
;       by Jean Meeus, p. 84 (Eq. 11-4) for the constants used.
;
; EXAMPLE:
;       Find the Greenwich mean sidereal time (GMST) on 2008 Jul 30 at 15:53 pm
;       in Baltimore, Maryland (longitude=-76.72 degrees).   The timezone is 
;       EDT or tz=-4
;
;       IDL> CT2LST, lst, -76.72, -4,ten(15,53), 30, 07, 2008
;
;               ==> lst =  11.356505  hours  (= 11h 21m 23.418s)
;
;       The Web site  http://tycho.usno.navy.mil/sidereal.html contains more
;       info on sidereal time, as well as an interactive calculator.
; PROCEDURES USED:
;       jdcnv - Convert from year, month, day, hour to julian date
;
; MODIFICATION HISTORY:
;     Adapted from the FORTRAN program GETSD by Michael R. Greason, STX, 
;               27 October 1988.
;     Use IAU 1984 constants Wayne Landsman, HSTX, April 1995, results 
;               differ by about 0.1 seconds  
;     Longitudes measured *east* of Greenwich   W. Landsman    December 1998
;     Time zone now measure positive East of Greenwich W. Landsman July 2008
;     Remove debugging print statement  W. Landsman April 2009
;-

*)

t0 := jd - jd2000;
t := t0/36525.0;
// Compute GST in seconds.
theta := 280.46061837 + (360.98564736629 * t0) + EXPT(t, 2)*(0.000387933 - (t/ 3871.0E4));
//theta := 100.46061837 + 36000.770053608*t0 + 0.000387933*EXPT(t0,2) - EXPT(t0,3)/3871000.0;
// Compute LST in hours.
CT2LST := ( theta + lng)/15.0;
CT2LST := MODABS(CT2LST, 24.0);

END_FUNCTION

// POUs/FUNCTIONS/DateTime2JD
FUNCTION DateTime2JD : LREAL
VAR_INPUT
	epoch			: TIMESTRUCT;
END_VAR
VAR
	a, y, m, d, jdn	: LREAL;
END_VAR

(*    import datetime
    from math import floor
    if not type(epoch) is datetime.datetime:
        raise TypeError('datetime must be of type datetime')
    
    a = floor((14 - epoch.month)/12)
    y = epoch.year + 4800 - a
    m = epoch.month + 12*a - 3
    
    d = epoch.day
    d += epoch.hour/24. + epoch.minute/1440. + epoch.second/86400. # microsecond might be added here?
    
    if [epoch.year,epoch.month,d] >= [1582,10,15]:
        jdn = epoch.day + floor((153*m + 2)/5) + 365*y + floor(y/4) - floor(y/100) + floor(y/400) - 32045
    elif [epoch.year,epoch.month,d] <= [1582,10,4]:
        jdn = epoch.day + floor((153*m + 2)/5) + 365*y + floor(y/4) - 32083
    return jdn + (epoch.hour-12)/24. + epoch.minute/1440. + epoch.second/86400.
*)
a := FLOOR((14.0 - epoch.wMonth)/12.0);
y := epoch.wYear + 4800.0 - a;
m := epoch.wMonth + 12.0*a - 3.0;

d := epoch.wDay + (epoch.wHour/24.0) + (epoch.wMinute/1440.0) + (epoch.wSecond/86400.0);

//IF (epoch.wYear > 1582) (* AND (epoch.wMonth > 10.0) AND (d > 15.0)*) THEN
	jdn := epoch.wDay + FLOOR((153*m + 2)/5) + 365.0*y + FLOOR(y/4) - FLOOR(y/100) + FLOOR(y/400) - 32045.0;
//ELSIF (epoch.wYear < 1582) AND (epoch.wMonth < 10) AND (d > 4.0) THEN
//	jdn := epoch.wDay + FLOOR((153*m + 2)/5) + 365.0*y + FLOOR(y/4) - 32083.0;
//END_IF

DateTime2JD := jdn
			+ (epoch.wHour-12.0)/24.0
			+ (epoch.wMinute/1440.0) 
			+ (epoch.wSecond/86400.0)
			+ (DWORD_TO_REAL(epoch.wMilliseconds)/86400000.0);

END_FUNCTION

// POUs/MAIN
PROGRAM MAIN
VAR
	estate 			: 	E_TestState := E_TestState.IDLE;	// different test states for the functions
	lat, lon        :   LREAL;							// location for observer						
	ra, dec			:   LREAL;							// coord eq
	alt, az			:   LREAL;							// coord eq
	eq2hor			:	FB_EQ2HOR;						// equatorial to horizontal transform function block (Stella1) (J2000) in degrees (FK5)
	hor2eq			:	FB_HOR2EQ;						// horizontal to equatorial transform function block (Stella1) (J2000) in degrees (FK5)
	
	lst1			: 	LREAL;
	jd1				:	LREAL;
	cycle_time		:	LREAL;
END_VAR

CASE estate OF
	E_TestState.IDLE:
		estate := E_TestState.IDLE;
		
		
	E_TestState.JD2LST:
		// transform time
		lst1 := JD2LST(jd := jd1, lon := lon);
		// return to IDLE
		cycle_time := UDINT_TO_LREAL(_TaskInfo[GETCURTASKINDEXEX()].CycleTime) / 10_000_000;
		estate := E_TestState.IDLE;
		
		
	E_TestState.EQ2HOR:
		// transform coordinates
		eq2hor(ra:=ra, dec:=dec, jd:=jd1, lon:=lon, lat:=lat, refract:=FALSE, alt=>alt, az=>az);
		// return to IDLE
		cycle_time := UDINT_TO_LREAL(_TaskInfo[GETCURTASKINDEXEX()].CycleTime) / 10_000_000;
		estate := E_TestState.IDLE;
	E_TestState.EQ2EQ:
		// transform to ALT AZ
		eq2hor(ra:=ra, dec:=dec, JD:=jd1, lon:=lon, lat:=lat, refract:=FALSE, alt=>alt, az=>az);
		// transform back :)
		hor2eq(alt:=alt, az:=az, jd:=jd1,lon:=lon, lat:=lat, refract:=FALSE, ra=>ra, dec=>dec);
		estate := E_TestState.IDLE;
	E_TestState.HOR2EQ:
		// transform :)
		hor2eq(alt:=alt, az:=az, jd:=jd1 , lon:=lon, lat:=lat, refract:=FALSE, ra=>ra, dec=>dec);
		estate := E_TestState.IDLE;
END_CASE

END_PROGRAM
